FUNCTION_BLOCK SDO_READ_FUNCTION_BLOCK
VAR_INPUT
	bExecute 					: 	BOOL;
	id							:	DINT;
END_VAR                     	
VAR_OUTPUT                  	
	value						:	REAL;
	qFmt						:	DINT;     
	bDone						:	BOOL;                   	
	bBusy 						: 	BOOL;
	bError						:	BOOL;
	nErrId						:	UDINT;
END_VAR
VAR
	CoeSdoRead 					:	FB_EcCoeSdoRead;
	CoeSdoWrite					:	FB_EcCoeSdoWrite;
	
	T_sNetID					:	T_AmsNetID;
	sNetID			AT%I*		:	AmsNetID;
	nSlaveAddr		AT%I*		:	UINT;
	nSubIndex					:	BYTE;
	nIndex						:	WORD;
	
	Buffer						:	ARRAY[0..2] OF DINT;
	
	state						:	INT	:= 0;
END_VAR

T_sNetid := CONCAT(BYTE_TO_STRING(sNetId[0]),'.');
T_sNetid := CONCAT(T_sNetId, BYTE_TO_STRING(sNetId[1]));	T_sNetid := CONCAT(T_sNetId,'.');
T_sNetid := CONCAT(T_sNetId, BYTE_TO_STRING(sNetId[2]));	T_sNetid := CONCAT(T_sNetId,'.');
T_sNetid := CONCAT(T_sNetId, BYTE_TO_STRING(sNetId[3]));	T_sNetid := CONCAT(T_sNetId,'.');
T_sNetid := CONCAT(T_sNetId, BYTE_TO_STRING(sNetId[4]));	T_sNetid := CONCAT(T_sNetId,'.');
T_sNetid := CONCAT(T_sNetId, BYTE_TO_STRING(sNetId[5]));
//temporary
//nSubIndex := 02;
nIndex := 16#2030;

//component trasformation
Buffer[0] := (SHL(16#02,24)+SHL(4,16)+SHL(id,8)+0);					//head of mailbox

IF NOT bExecute THEN
	state := 0;
END_IF

CASE state OF
0://initialization
	CoeSdoRead(bExecute:=FALSE);
	CoeSdoWrite(bExecute:=FALSE);
	
	bDone := FALSE;
	bBusy := FALSE;
	bError := FALSE;
	nErrId := 0;
	
	IF bExecute THEN
		state := 10;
	END_IF
	
10://write headword
	bDone := FALSE;
	bBusy := TRUE;
	bError := FALSE;
	nErrId := 0;
	
	CoeSdoWrite(
		sNetId:= T_sNetId, 
		nSlaveAddr:= nSlaveAddr, 
		nSubIndex:= 01, 
		nIndex:= nIndex, 
		pSrcBuf:= ADR(Buffer[0]), 
		cbBufLen:= SIZEOF(Buffer[0]), 
		bExecute:= TRUE, 
		bBusy=> , 
		bError=> , 
		nErrId=> );
		
	IF NOT CoeSdoWrite.bBusy AND NOT CoeSdoWrite.bError THEN
		CoeSdoWrite(bExecute:=FALSE);
		state := 20;
	ELSIF CoeSdoWrite.bError THEN
		nErrId := CoeSdoWrite.nErrId;
		bError := TRUE;
	END_IF

20://read value
	CoeSdoRead(
		sNetId:= T_sNetID, 
		nSlaveAddr:= nSlaveAddr, 
		nSubIndex:= 02, 
		nIndex:= nIndex, 
		pDstBuf:= ADR(Buffer[1]), 
		cbBufLen:= SIZEOF(Buffer[1]), 
		bExecute:= TRUE, 
		bBusy=> , 
		bError=> , 
		nErrId=> );
		
	IF NOT CoeSdoRead.bBusy AND NOT CoeSdoRead.bError THEN
		CoeSdoRead(bExecute:=FALSE);
		state := 30;
	ELSIF CoeSdoRead.bError THEN
		nErrId := CoeSdoRead.nErrId;
		bError := TRUE;
	END_IF
	
30://read q-value
	CoeSdoRead(
		sNetId:= T_sNetID, 
		nSlaveAddr:= nSlaveAddr, 
		nSubIndex:= 03, 
		nIndex:= nIndex, 
		pDstBuf:= ADR(Buffer[2]), 
		cbBufLen:= SIZEOF(Buffer[2]), 
		bExecute:= TRUE, 
		tTimeout:= , 
		bBusy=> ,
		bError=> , 
		nErrId=> );
	IF NOT CoeSdoRead.bBusy AND NOT CoeSdoRead.bError THEN
		CoeSdoWrite(bExecute:=FALSE);
		state := 40;
	ELSIF CoeSdoRead.bError THEN
		nErrId := CoeSdoWrite.nErrId;
		bError := TRUE;
	END_IF
	
40:
	qFmt := Buffer[2];	
	value := DINT_TO_REAL(Buffer[1])/EXPT(10,qFmt);

	bDone := TRUE;
	bBusy := FALSE;
	bError := FALSE;
	nErrId := 0;
END_CASE

END_FUNCTION_BLOCK

(* stored: Version 1.1.0.1, ProductVersion 3.1.4020.12
   POU SDO_READ_FUNCTION_BLOCK: Id {a50fcd84-3936-46da-ada2-6d366663847a}, SpecialFunc None *)
